{attribute 'qualified_only'}
{attribute 'strict'}
TYPE eState :
(
	Undefine	:= -1,
	PowerOff	:= 0,
	Home		:= 1,
	Ready		:= 2,
	Running		:= 3,
	Alarm		:= 4,
	Emptying	:= 5,
	Loading		:= 6,
	Manual		:= 7,
	UpsOn		:= 99 //solo per database, creato internamente in PLC Beckhoff
);
END_TYPE
//  Undefine = '-1'

(* stored: Version 1.1.0.1, ProductVersion 3.1.4024.15
   EnumerationTextList eState: Id {28718a8c-b176-4530-a98c-2cc4e088b232} *)
